{attribute 'qualified_only'}
//{attribute 'strict'}
{attribute 'to_string'}

TYPE E_Stop_Cmds :
(
	Reset :=0,
	Stop_Cycle,
	Shutdown_Safe,
	Shutdown_Evac,
	Estop
);
END_TYPE

(* stored: Version 1.1.0.1, ProductVersion 3.1.4024.12
   DUT E_Stop_Cmds: Id {2053f432-3167-47c9-9b78-33b40257e7a8} *)
